# EPICS substitutions: iocBoot/iocnamWin/substitutions/canberra_3.substitutions
file "$(MCA)/mcaApp/Db/simple_mca.db"
{
pattern
{P           M       DTYP           INP              PREC  CHANS}
{namWin:med:   mca1  "asynMCA"       "@asyn(AIM1/1 0)"  3     2048}
{namWin:med:   mca2  "asynMCA"       "@asyn(AIM1/2 0)"  3     2048}
{namWin:med:   mca3  "asynMCA"       "@asyn(AIM2/1 0)"  3     2048}
{namWin:med:   mca0  "Soft Channel"  ""                 3     2048}
}

#file "$(MCA)/mcaApp/Db/icb_amp.db"
#{
#pattern
#{P			AMP		PORT}
#{namWin:med:	amp1	icbAmp1}
#}

file "$(MCA)/mcaApp/Db/icb_adc.db"
{
pattern
{P			ADC		PORT}
{namWin:med:	adc1	"icbAdc1"}
{namWin:med:	adc2	"icbAdc2"}
{namWin:med:	adc3	"icbAdc3"}
}

#file "$(MCA)/mcaApp/Db/icb_hvps.db"
#{
#pattern
#{P			HVPS	LIMIT	PORT}
#{namWin:med:	hvps1	1000	"icbHvps1"}
#}

file "$(MCA)/mcaApp/Db/icb_tca.db"
{
pattern
{P,          TCA,	PORT,		MCA}
{namWin:med:,  tca1,	"icbTca1",	mca1}
{namWin:med:,  tca2,	"icbTca2",	mca2}
{namWin:med:,  tca3,	"icbTca3",	mca3}
}
